{attribute addProperty BoxType "EL5001-0000-1021"}
{attribute addProperty Id "SSI_InputsAT %I*SSI_Inputs_B703DF694860WcStateAT %I*WcState_F855686C1620InfoDataAT %I*InfoData_BC63D37F80100"}
{attribute addProperty CRC "4051780250"}
{attribute addProperty SizeInBites "144"}
{attribute addProperty SizeInBytes "18"}
TYPE EL5001_F220A1B7 :
STRUCT
	{attribute addProperty Name "SSI_Inputs"}
	SSI_Inputs : SSI_Inputs_B703DF69;
	{attribute addProperty Name "WcState"}
	WcState : WcState_F855686C;
	{attribute addProperty Name "InfoData"}
	InfoData : InfoData_BC63D37F;
END_STRUCT
END_TYPE

(* stored: Version 1.2.0.0, ProductVersion 3.1.4024.9
   DUT EL5001_F220A1B7: Id {7e9f8e78-a3c8-4f8c-b547-3933e3e23557} *)
